(* PLC project  *)

FUNCTION_BLOCK SR
  VAR_INPUT
    S1 : BOOL;
    R : BOOL;
  END_VAR
  VAR_OUTPUT
    Q1 : BOOL;
  END_VAR
  VAR
    Q1 : BOOL;
  END_VAR

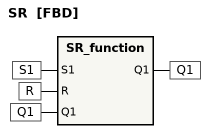
(* FBD diagram, written out as Structured Text *)
Q1 := SR_function(S1, R, Q1);
END_FUNCTION_BLOCK

FUNCTION_BLOCK RS
  VAR_INPUT
    S : BOOL;
    R1 : BOOL;
  END_VAR
  VAR_OUTPUT
    Q1 : BOOL;
  END_VAR
  VAR
    Q1 : BOOL;
  END_VAR

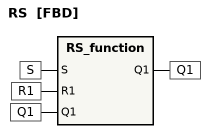
(* FBD diagram, written out as Structured Text *)
Q1 := RS_function(S, R1, Q1);
END_FUNCTION_BLOCK

FUNCTION_BLOCK CTU
  VAR_INPUT
    CU : BOOL;
    R : BOOL;
    PV : INT;
  END_VAR
  VAR_OUTPUT
    Q : BOOL;
    CV : INT;
  END_VAR
  VAR
    CV : INT;
    TRIG_M : BOOL;
  END_VAR
  VAR  (* added by the conversion: wires and edge detectors of the diagram *)
    _CTU_function7_CV : ANY;
    _CTU_function7_TRIG_M : ANY;
    _CTU_function7_OUT : BOOL;
  END_VAR

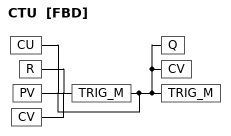
(* FBD diagram, written out as Structured Text *)
_CTU_function7_OUT := CTU_function(CU := CU, R := R, PV := PV, CV := CV, TRIG_M := TRIG_M, CV => _CTU_function7_CV, TRIG_M => _CTU_function7_TRIG_M);
Q := TRIG_M;
CV := TRIG_M;
TRIG_M := TRIG_M;
END_FUNCTION_BLOCK

FUNCTION_BLOCK CTD
  VAR_INPUT
    CD : BOOL;
    LD : BOOL;
    PV : INT;
  END_VAR
  VAR_OUTPUT
    Q : BOOL;
    CV : INT;
  END_VAR
  VAR
    CV : INT;
    TRIG_M : BOOL;
  END_VAR
  VAR  (* added by the conversion: wires and edge detectors of the diagram *)
    _CTD_function7_CV : ANY;
    _CTD_function7_OUT : BOOL;
  END_VAR

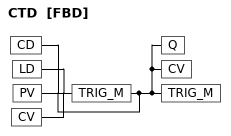
(* FBD diagram, written out as Structured Text *)
_CTD_function7_OUT := CTD_function(CD := CD, LD := LD, PV := PV, CV := CV, TRIG_M := TRIG_M, CV => _CTD_function7_CV);
Q := TRIG_M;
CV := TRIG_M;
TRIG_M := TRIG_M;
END_FUNCTION_BLOCK

FUNCTION_BLOCK CTUD
  VAR_INPUT
    CU : BOOL;
    CD : BOOL;
    R : BOOL;
    LD : BOOL;
    PV : INT;
  END_VAR
  VAR_OUTPUT
    QU : BOOL;
    QD : BOOL;
    CV : INT;
  END_VAR
  VAR
    CV : INT;
    TRIG_MU : BOOL;
    TRIG_MD : BOOL;
  END_VAR
  VAR  (* added by the conversion: wires and edge detectors of the diagram *)
    _CTUD_function7_QD : ANY;
    _CTUD_function7_CV : ANY;
    _CTUD_function7_OUT : BOOL;
  END_VAR

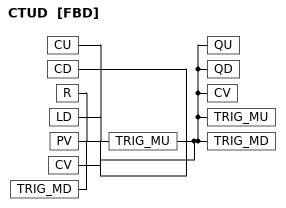
(* FBD diagram, written out as Structured Text *)
_CTUD_function7_OUT := CTUD_function(CU := CU, CD := CD, R := R, LD := LD, PV := PV, CV := CV, TRIG_MU := TRIG_MU, TRIG_MD := TRIG_MD, QD => _CTUD_function7_QD, CV => _CTUD_function7_CV);
QU := TRIG_MU;
QD := TRIG_MU;
CV := TRIG_MU;
TRIG_MU := TRIG_MU;
TRIG_MD := TRIG_MU;
END_FUNCTION_BLOCK

FUNCTION_BLOCK R_TRIG
  VAR_INPUT
    CLK : BOOL;
  END_VAR
  VAR_OUTPUT
    Q : BOOL;
  END_VAR
  VAR
    M : BOOL;
  END_VAR
  VAR  (* added by the conversion: wires and edge detectors of the diagram *)
    _R_TRIG_function7_M : ANY;
    _R_TRIG_function7_OUT : BOOL;
  END_VAR

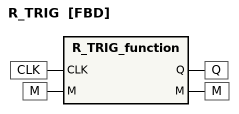
(* FBD diagram, written out as Structured Text *)
_R_TRIG_function7_OUT := R_TRIG_function(CLK := CLK, M := M, M => _R_TRIG_function7_M);
Q := _R_TRIG_function7_OUT;
M := _R_TRIG_function7_M;
END_FUNCTION_BLOCK

FUNCTION_BLOCK F_TRIG
  VAR_INPUT
    CLK : BOOL;
  END_VAR
  VAR_OUTPUT
    Q : BOOL;
  END_VAR
  VAR
    M : BOOL;
  END_VAR
  VAR  (* added by the conversion: wires and edge detectors of the diagram *)
    _F_TRIG_function7_M : ANY;
    _F_TRIG_function7_OUT : BOOL;
  END_VAR

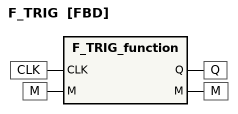
(* FBD diagram, written out as Structured Text *)
_F_TRIG_function7_OUT := F_TRIG_function(CLK := CLK, M := M, M => _F_TRIG_function7_M);
Q := _F_TRIG_function7_OUT;
M := _F_TRIG_function7_M;
END_FUNCTION_BLOCK

FUNCTION_BLOCK RTC
  VAR_INPUT
    IN : BOOL;
    PDT : DT;
  END_VAR
  VAR_OUTPUT
    Q : BOOL;
    CDT : DT;
  END_VAR
  VAR
    PREV_IN : BOOL;
    OFFSET : TIME;
  END_VAR
  VAR  (* added by the conversion: wires and edge detectors of the diagram *)
    _RTC_function7_CDT : ANY;
    _RTC_function7_PREV_IN : ANY;
    _RTC_function7_OFFSET : ANY;
    _RTC_function7_OUT : BOOL;
  END_VAR

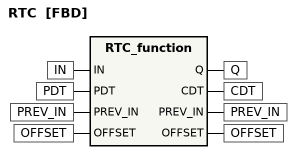
(* FBD diagram, written out as Structured Text *)
_RTC_function7_OUT := RTC_function(IN := IN, PDT := PDT, PREV_IN := PREV_IN, OFFSET := OFFSET, CDT => _RTC_function7_CDT, PREV_IN => _RTC_function7_PREV_IN, OFFSET => _RTC_function7_OFFSET);
Q := _RTC_function7_OUT;
CDT := _RTC_function7_CDT;
PREV_IN := _RTC_function7_PREV_IN;
OFFSET := _RTC_function7_OFFSET;
END_FUNCTION_BLOCK

FUNCTION_BLOCK TP
  VAR_INPUT
    IN : BOOL;
    PT : TIME;
  END_VAR
  VAR_OUTPUT
    Q : BOOL;
    ET : TIME;
  END_VAR
  VAR
    STATE : SINT;
    PREV_IN : BOOL;
    START_TIME : TIME;
    Q : BOOL;
    ET : TIME;
  END_VAR
  VAR  (* added by the conversion: wires and edge detectors of the diagram *)
    _TP_function7_OUT : ANY;
    _TP_function7_ET : ANY;
    _TP_function7_STATE : ANY;
    _TP_function7_PREV_IN : ANY;
    _TP_function7_START_TIME : ANY;
  END_VAR

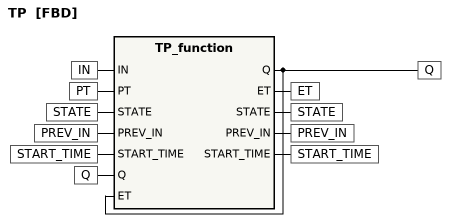
(* FBD diagram, written out as Structured Text *)
_TP_function7_OUT := TP_function(IN := IN, PT := PT, STATE := STATE, PREV_IN := PREV_IN, START_TIME := START_TIME, Q := Q, ET := _TP_function7_OUT, ET => _TP_function7_ET, STATE => _TP_function7_STATE, PREV_IN => _TP_function7_PREV_IN, START_TIME => _TP_function7_START_TIME);
Q := _TP_function7_OUT;
ET := _TP_function7_ET;
STATE := _TP_function7_STATE;
PREV_IN := _TP_function7_PREV_IN;
START_TIME := _TP_function7_START_TIME;
END_FUNCTION_BLOCK

FUNCTION_BLOCK TON
  VAR_INPUT
    IN : BOOL;
    PT : TIME;
  END_VAR
  VAR_OUTPUT
    Q : BOOL;
    ET : TIME;
  END_VAR
  VAR
    STATE : SINT;
    PREV_IN : BOOL;
    START_TIME : TIME;
    Q : BOOL;
    ET : TIME;
  END_VAR
  VAR  (* added by the conversion: wires and edge detectors of the diagram *)
    _TON_function7_OUT : ANY;
    _TON_function7_ET : ANY;
    _TON_function7_STATE : ANY;
    _TON_function7_PREV_IN : ANY;
    _TON_function7_START_TIME : ANY;
  END_VAR

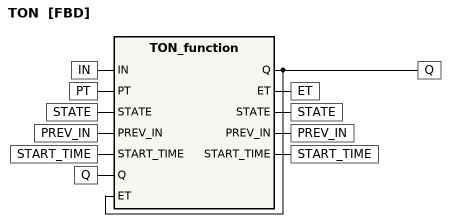
(* FBD diagram, written out as Structured Text *)
_TON_function7_OUT := TON_function(IN := IN, PT := PT, STATE := STATE, PREV_IN := PREV_IN, START_TIME := START_TIME, Q := Q, ET := _TON_function7_OUT, ET => _TON_function7_ET, STATE => _TON_function7_STATE, PREV_IN => _TON_function7_PREV_IN, START_TIME => _TON_function7_START_TIME);
Q := _TON_function7_OUT;
ET := _TON_function7_ET;
STATE := _TON_function7_STATE;
PREV_IN := _TON_function7_PREV_IN;
START_TIME := _TON_function7_START_TIME;
END_FUNCTION_BLOCK

FUNCTION_BLOCK TOF
  VAR_INPUT
    IN : BOOL;
    PT : TIME;
  END_VAR
  VAR_OUTPUT
    Q : BOOL;
    ET : TIME;
  END_VAR
  VAR
    STATE : SINT;
    PREV_IN : BOOL;
    START_TIME : TIME;
  END_VAR
  VAR  (* added by the conversion: wires and edge detectors of the diagram *)
    _TOF_function7_ET : ANY;
    _TOF_function7_STATE : ANY;
    _TOF_function7_PREV_IN : ANY;
    _TOF_function7_START_TIME : ANY;
    _TOF_function7_OUT : BOOL;
  END_VAR

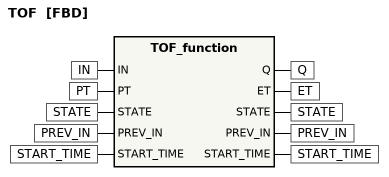
(* FBD diagram, written out as Structured Text *)
_TOF_function7_OUT := TOF_function(IN := IN, PT := PT, STATE := STATE, PREV_IN := PREV_IN, START_TIME := START_TIME, ET => _TOF_function7_ET, STATE => _TOF_function7_STATE, PREV_IN => _TOF_function7_PREV_IN, START_TIME => _TOF_function7_START_TIME);
Q := _TOF_function7_OUT;
ET := _TOF_function7_ET;
STATE := _TOF_function7_STATE;
PREV_IN := _TOF_function7_PREV_IN;
START_TIME := _TOF_function7_START_TIME;
END_FUNCTION_BLOCK

FUNCTION_BLOCK HYSTERESIS
  VAR_INPUT
    XIN1 : REAL;
    XIN2 : REAL;
    EPS : REAL;
  END_VAR
  VAR_OUTPUT
    Q : BOOL;
  END_VAR
  VAR
    Q : BOOL;
  END_VAR

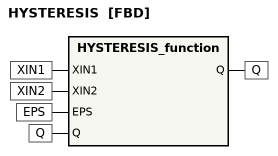
(* FBD diagram, written out as Structured Text *)
Q := HYSTERESIS_function(XIN1, XIN2, EPS, Q);
END_FUNCTION_BLOCK

FUNCTION_BLOCK DERIVATIVE
  VAR_INPUT
    RUN : BOOL;
    XIN : REAL;
    CYCLE : TIME;
  END_VAR
  VAR_OUTPUT
    XOUT : REAL;
  END_VAR
  VAR
    X1 : DINT;
    X2 : DINT;
    X3 : DINT;
  END_VAR
  VAR  (* added by the conversion: wires and edge detectors of the diagram *)
    _DERIVATIVE_function100_X1 : ANY;
    _DERIVATIVE_function100_X2 : ANY;
    _DERIVATIVE_function100_X3 : ANY;
    _DERIVATIVE_function100_OUT : BOOL;
  END_VAR

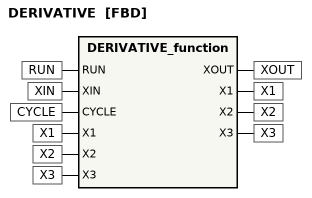
(* FBD diagram, written out as Structured Text *)
_DERIVATIVE_function100_OUT := DERIVATIVE_function(RUN := RUN, XIN := XIN, CYCLE := CYCLE, X1 := X1, X2 := X2, X3 := X3, X1 => _DERIVATIVE_function100_X1, X2 => _DERIVATIVE_function100_X2, X3 => _DERIVATIVE_function100_X3);
XOUT := _DERIVATIVE_function100_OUT;
X1 := _DERIVATIVE_function100_X1;
X2 := _DERIVATIVE_function100_X2;
X3 := _DERIVATIVE_function100_X3;
END_FUNCTION_BLOCK
